// TIA Portal V20 export
TYPE "LER_typeAxisInterlock"
// stored: Access Published
   STRUCT
      permit : "LER_typeAxisInterlockPermit";
      source : "LER_typeAxisInterlockSource";
   END_STRUCT;
END_TYPE
